FUNCTION_BLOCK ABSTRACT FB_AltAzTelescopeControl EXTENDS FB_BaseTelescopeControl IMPLEMENTS I_AltAzTelescope
VAR_INPUT
	fElevationOffset	: LREAL := 0.0;		// absolute offset for elevation
	fAzimuthOffset 		: LREAL := 0.0;		// absolute offset for azimuth
	fDerotatorOffset	: LREAL := 0.0;		// offset for the de-rotator
	// UT1-UTC (seconds, IERS). 0.0 = treat UTC as UT1 (no correction), matching FB_EQ2HOR/
	// FB_HOR2EQ's own default. Set via MQTT by an external time bridge (Dut1 property, see
	// FB_Comm_MQTT_Influx); reverts to 0.0 if nothing fresh arrives for a while (below).
	fDut1				: LREAL := 0.0;
END_VAR
VAR_OUTPUT
	fDerotatorCurrent	: LREAL;	// current position in derotator (calculated) (without pointing and offset correction)
END_VAR
VAR
	eq2hor				: FB_EQ2HOR;
	hor2eq				: FB_HOR2EQ;

	fDerotatorCalc		: LREAL;	// derotator angle calcuilated

	bDut1Received		: BOOL;
	tonDut1Stale		: TON := (PT := T#10M);
END_VAR
// The pointing-model coefficients live in FB_PointingModelForward, set by the caller (#10).

SUPER^();

METHOD _PublishTelemetry : BOOL
VAR_INPUT
END_VAR
SUPER^._PublishTelemetry();

fbComm.Publish('telescope', 'dome', 'POSITION.INSTRUMENTAL.AZ.OFFSET', LREAL_TO_STRING(fAzimuthOffset));
fbComm.Publish('telescope', 'dome', 'POSITION.INSTRUMENTAL.ALT.OFFSET', LREAL_TO_STRING(fElevationOffset));
END_METHOD

PROPERTY AltitudeOffset : LREAL
GET
AltitudeOffset := THIS^.fElevationOffset;
END_GET
SET
THIS^.fElevationOffset := AltitudeOffset;
END_SET
END_PROPERTY

PROPERTY AzimuthOffset : LREAL
GET
AzimuthOffset := THIS^.fAzimuthOffset;
END_GET
SET
THIS^.fAzimuthOffset := AzimuthOffset;
END_SET
END_PROPERTY

PROPERTY DerotatorOffset : LREAL
GET
DerotatorOffset := THIS^.fDerotatorOffset;
END_GET
SET
THIS^.fDerotatorOffset := DerotatorOffset;
END_SET
END_PROPERTY

PROPERTY Dut1 : LREAL
GET
Dut1 := THIS^.fDut1;
END_GET
SET
THIS^.fDut1 := Dut1;
THIS^.bDut1Received := TRUE;
END_SET
END_PROPERTY

END_FUNCTION_BLOCK

(* stored: Version 1.1.0.1, ProductVersion 3.1.4024.15
   POU FB_AltAzTelescopeControl: Id {ab7ff9f6-f0dc-473a-bd67-87367819c272}, SpecialFunc None
   Method _PublishTelemetry: Id {313bc6a7-19ec-4722-9d6e-3ac84aa9588f}
   Property AltitudeOffset: Id {61d61b42-3772-48a4-bbf4-c8264f7b8459}
   Get Get: Id {8a20eda7-7b14-4b00-8989-4e306a01fc43}
   Set Set: Id {1c47573f-0f89-4ecb-9bcf-d7511a1c4e19}
   Property AzimuthOffset: Id {580c6b01-71eb-41a5-b2e8-f0166c9039a8}
   Get Get: Id {ed413719-73e2-4660-85da-efe3c363e7f1}
   Set Set: Id {732d8f9f-01ec-4777-918f-f8df92d2605e}
   Property DerotatorOffset: Id {da6437af-965e-40c2-8dea-4bf926c328a7}
   Get Get: Id {340a3d36-9a30-422a-ad59-6bebfad8b2af}
   Set Set: Id {647130f3-7273-4691-ba3d-1e20d8a7157d}
   Property Dut1: Id {d1e2f3a4-5b6c-47d8-a9e0-1f2a3b4c5d6e}
   Get Get: Id {e2f3a4b5-6c7d-48e9-ba01-2f3a4b5c6d7e}
   Set Set: Id {f3a4b5c6-7d8e-49fa-cb12-3a4b5c6d7e8f} *)
